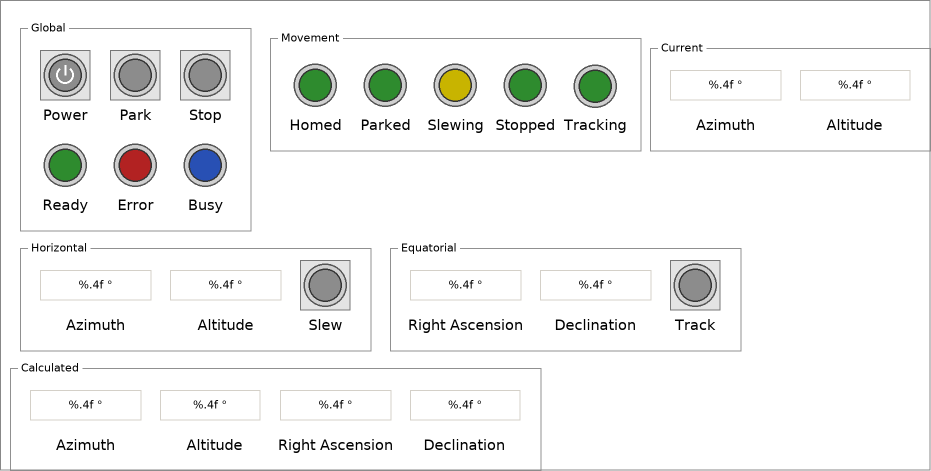
VISUALIZATION Telescope  // 931x471
    GroupBox (20,20 231x211), "Global"
        Label (0,80 91x30), "Power"
        Lamp1 (90,120 50x50), variable: MAIN.TelescopeControl.bError, style: Lamp-Lamp1-Red
        Label (90,170 51x30), "Error"
        Lamp1 (20,120 50x50), variable: MAIN.TelescopeControl.bReady, style: Lamp-Lamp1-Green
        Label (20,170 51x30), "Ready"
        PowerSwitch (20,30 50x50), variable: MAIN.TelescopeControl.bPower, behaviour: TOGGLE, style: Switch-PowerSwitch-Gray
        PushSwitch (90,30 50x50), variable: MAIN.TelescopeControl.bPark, behaviour: TOGGLE, style: Switch-PushSwitch-Gray
        Lamp1 (160,120 50x50), variable: MAIN.TelescopeControl.bBusy, style: Lamp-Lamp1-Blue
        Label (160,170 51x30), "Busy"
        PushSwitch (160,30 50x50), variable: MAIN.TelescopeControl.bPark, behaviour: TOGGLE, style: Switch-PushSwitch-Gray
        Label (140,80 91x30), "Stop"
    Label (90,100 91x30), "Park"
    GroupBox (20,240 351x111), "Horizontal"
        Label (30,70 91x30), "Azimuth"
        Textfield (20,30 111x30), "%.4f °", text variable: MAIN.TelescopeControl.fAzimuth
            OnMouseClick: write the text variable via InputWithLimits, min 0, max 360
        Label (160,70 91x30), "Altitude"
        PushSwitch (280,20 50x50), variable: MAIN.TelescopeControl.bSlew, behaviour: TOGGLE, style: Switch-PushSwitch-Gray
        Label (260,70 91x30), "Slew"
    Textfield (170,270 111x30), "%.4f °", text variable: MAIN.TelescopeControl.fElevation
        OnMouseClick: write the text variable via Default, min 0, max 90
    GroupBox (10,360 531x111), "Calculated"
        Label (30,70 91x30), "Azimuth"
        Textfield (20,30 111x30), "%.4f °", text variable: MAIN.TelescopeControl.fAzimuthCalc
        Label (159,70 91x30), "Altitude"
        Textfield (150,30 100x30), "%.4f °", text variable: MAIN.TelescopeControl.fElevationCalc
        Label (270,70 111x30), "Right Ascension"
        Textfield (270,30 111x30), "%.4f °", text variable: MAIN.TelescopeControl.fRightAscensionCalc
        Label (409,70 91x30), "Declination"
        Textfield (400,30 110x30), "%.4f °", text variable: MAIN.TelescopeControl.fDeclinationCalc
    GroupBox (650,40 281x111), "Current"
        Label (30,70 91x30), "Azimuth"
        Textfield (20,30 111x30), "%.4f °", text variable: MAIN.TelescopeControl.fAzimuthCurrent
        Label (159,70 91x30), "Altitude"
        Textfield (150,30 110x30), "%.4f °", text variable: MAIN.TelescopeControl.fElevationCurrent
    GroupBox (270,30 371x121), "Movement"
        Lamp1 (90,30 50x50), variable: MAIN.TelescopeControl.isparked, style: Lamp-Lamp1-Green
        Label (90,80 51x30), "Parked"
        Lamp1 (160,30 50x50), variable: MAIN.TelescopeControl.bSlewing, style: Lamp-Lamp1-Yellow
        Label (150,80 71x30), "Slewing"
        Lamp1 (230,30 50x50), variable: MAIN.TelescopeControl.bStopped, style: Lamp-Lamp1-Green
        Label (220,80 71x30), "Stopped"
        Lamp1 (300,31 50x50), variable: MAIN.TelescopeControl.bTracking, style: Lamp-Lamp1-Green
        Label (290,80 71x30), "Tracking"
        Lamp1 (20,30 50x50), variable: MAIN.TelescopeControl.bHomed, style: Lamp-Lamp1-Green
        Label (20,80 51x30), "Homed"
    GroupBox (390,240 351x111), "Equatorial"
        Label (20,70 111x30), "Right Ascension"
        Textfield (20,30 111x30), "%.4f °", text variable: MAIN.TelescopeControl.fRightAscension
            OnMouseClick: write the text variable via InputWithLimits, min 0, max 360
        Label (160,70 91x30), "Declination"
        PushSwitch (280,20 50x50), variable: MAIN.TelescopeControl.bGoto, behaviour: TOGGLE, style: Switch-PushSwitch-Gray
        Label (260,70 91x30), "Track"
        Textfield (150,30 111x30), "%.4f °", text variable: MAIN.TelescopeControl.fDeclination
            OnMouseClick: write the text variable via Default, min -90, max 90
END_VISUALIZATION

(* stored: Version 1.1.0.1, ProductVersion 3.1.4024.15
   Visu Telescope: Id {6ed16cb5-124e-425d-aa65-71916eed16eb} *)
